// Mitsubishi GX Works2 project: 241108_PLC_PRACTICE3   PLC: Q02U

PROGRAM MAIN
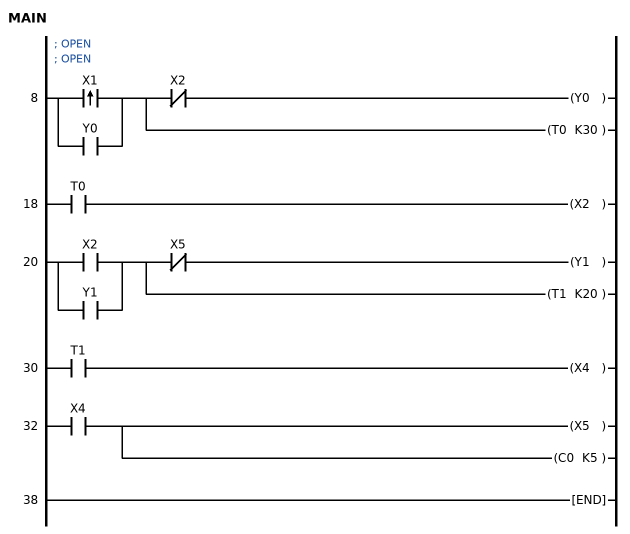
; OPEN
; OPEN
8     LDP     X1
      OR      Y0
      MPS
      ANI     X2
      OUT     Y0
      MPP
      OUT     T0 K30
18    LD      T0
      OUT     X2
20    LD      X2
      OR      Y1
      MPS
      ANI     X5
      OUT     Y1
      MPP
      OUT     T1 K20
30    LD      T1
      OUT     X4
32    LD      X4
      OUT     X5
      OUT     C0 K5
38    END
END_PROGRAM
